FUNCTION_BLOCK DAerationLogicBasic (* Basic Function Block Type *)
  (* Standard: 61499-2 *)
  (* Version 0.0, 6/10/2026, Schneider Electric, Template *)
  PACKAGE SE.Nereda;
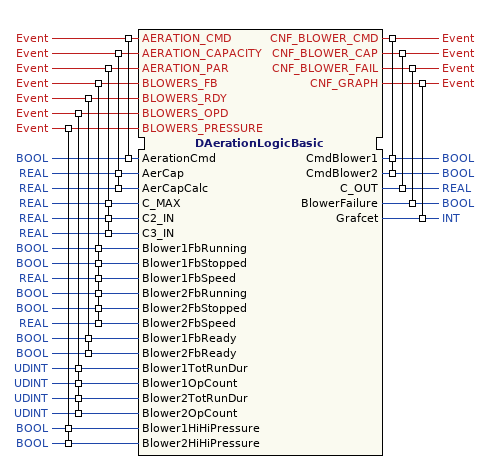
  EVENT_INPUT
    AERATION_CMD WITH AerationCmd;
    AERATION_CAPACITY WITH AerCap, AerCapCalc;
    AERATION_PAR WITH C_MAX, C2_IN, C3_IN;
    BLOWERS_FB WITH Blower1FbRunning, Blower1FbStopped, Blower1FbSpeed, Blower2FbRunning, Blower2FbStopped, Blower2FbSpeed;
    BLOWERS_RDY WITH Blower1FbReady, Blower2FbReady;
    BLOWERS_OPD WITH Blower1TotRunDur, Blower2TotRunDur, Blower1OpCount, Blower2OpCount;
    BLOWERS_PRESSURE WITH Blower1HiHiPressure, Blower2HiHiPressure;
  END_EVENT
  EVENT_OUTPUT
    CNF_BLOWER_CMD WITH CmdBlower1, CmdBlower2;
    CNF_BLOWER_CAP WITH C_OUT;
    CNF_BLOWER_FAIL WITH BlowerFailure;
    CNF_GRAPH WITH Grafcet;
  END_EVENT
  VAR_INPUT
    AerationCmd : BOOL;
    AerCap : REAL;
    AerCapCalc : REAL;
    C_MAX : REAL;
    C2_IN : REAL;
    C3_IN : REAL;
    Blower1FbRunning : BOOL;
    Blower1FbStopped : BOOL;
    Blower1FbSpeed : REAL;
    Blower2FbRunning : BOOL;
    Blower2FbStopped : BOOL;
    Blower2FbSpeed : REAL;
    Blower1FbReady : BOOL;
    Blower2FbReady : BOOL;
    Blower1TotRunDur : UDINT;
    Blower1OpCount : UDINT;
    Blower2TotRunDur : UDINT;
    Blower2OpCount : UDINT;
    Blower1HiHiPressure : BOOL;
    Blower2HiHiPressure : BOOL;
  END_VAR
  VAR_OUTPUT
    CmdBlower1 : BOOL;
    CmdBlower2 : BOOL;
    C_OUT : REAL;
    BlowerFailure : BOOL;
    Grafcet : INT;
  END_VAR
  VAR
    BL1WasRun : BOOL;
    BL2WasRun : BOOL;
  END_VAR
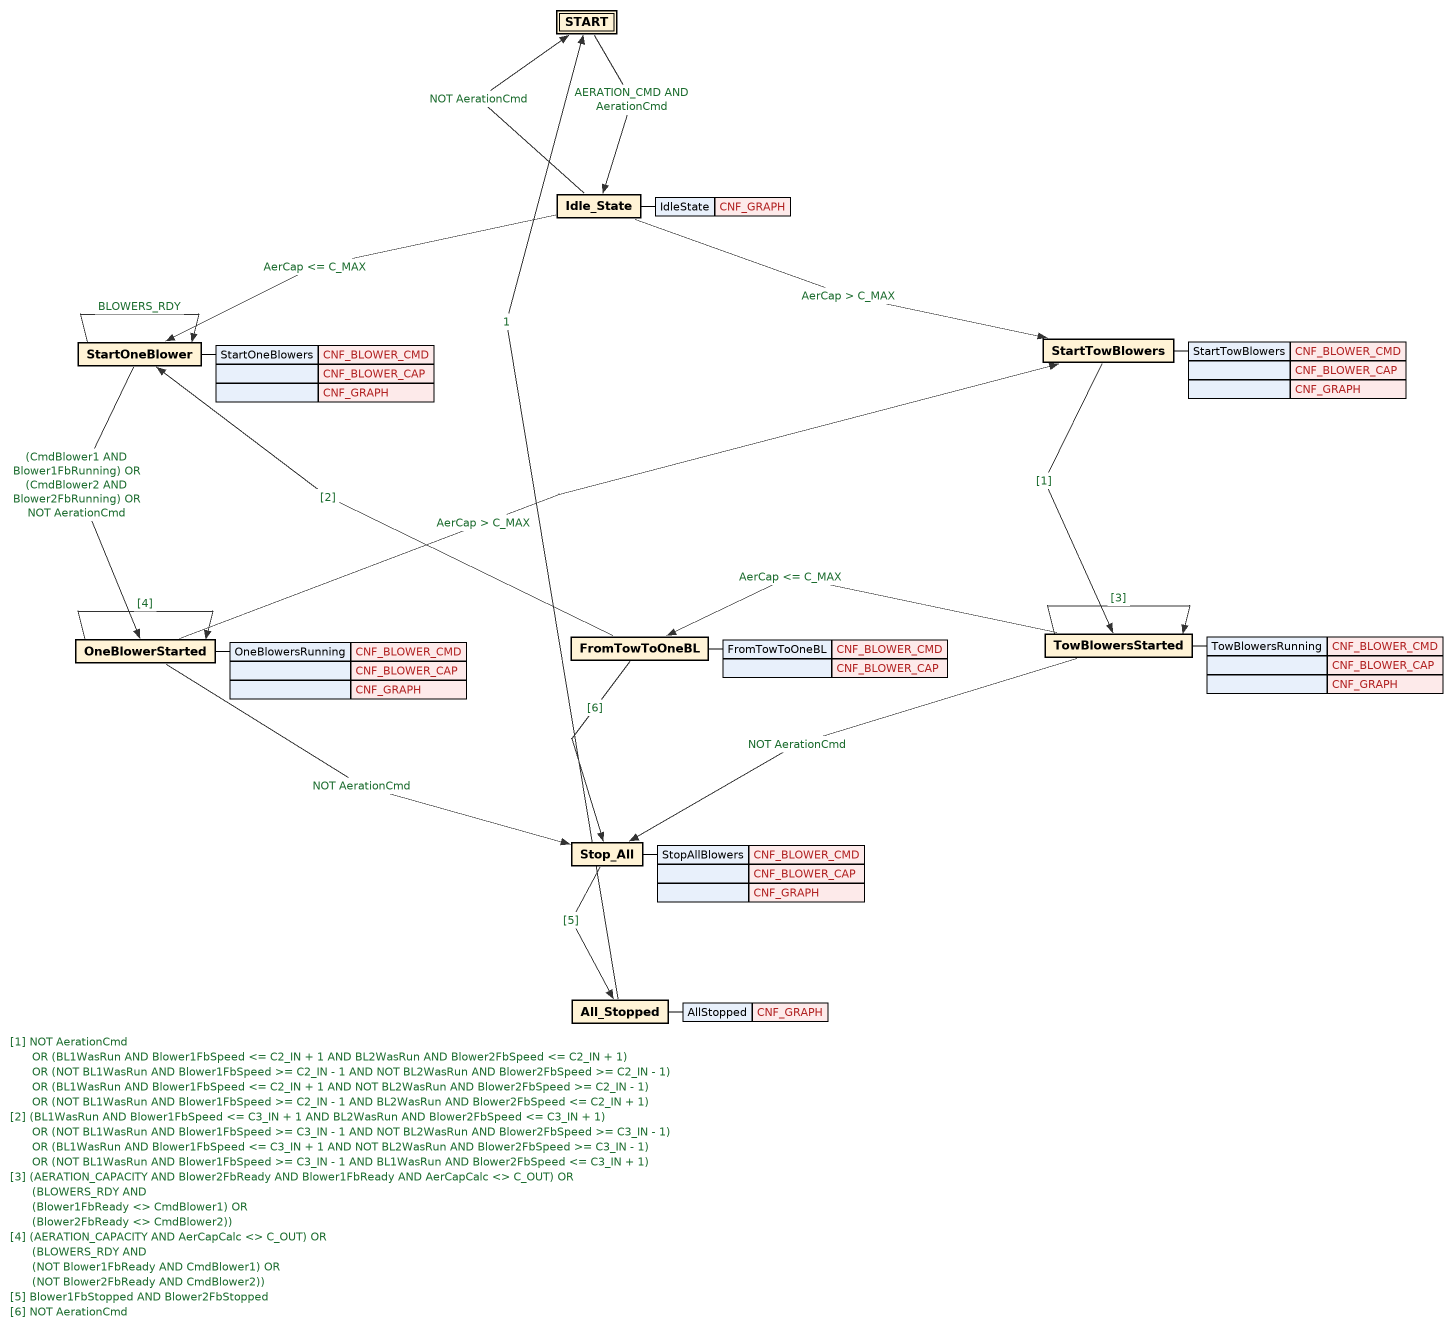
  EC_STATES
    START; (* Initial State *)
    Idle_State : IdleState -> CNF_GRAPH;
    StartTowBlowers : StartTowBlowers -> CNF_BLOWER_CMD, -> CNF_BLOWER_CAP, -> CNF_GRAPH;
    StartOneBlower : StartOneBlowers -> CNF_BLOWER_CMD, -> CNF_BLOWER_CAP, -> CNF_GRAPH;
    OneBlowerStarted : OneBlowersRunning -> CNF_BLOWER_CMD, -> CNF_BLOWER_CAP, -> CNF_GRAPH;
    TowBlowersStarted : TowBlowersRunning -> CNF_BLOWER_CMD, -> CNF_BLOWER_CAP, -> CNF_GRAPH;
    Stop_All : StopAllBlowers -> CNF_BLOWER_CMD, -> CNF_BLOWER_CAP, -> CNF_GRAPH;
    All_Stopped : AllStopped -> CNF_GRAPH;
    FromTowToOneBL : FromTowToOneBL -> CNF_BLOWER_CMD, -> CNF_BLOWER_CAP;
  END_STATES
  EC_TRANSITIONS
    START TO Idle_State := AERATION_CMD AND AerationCmd;
    Idle_State TO StartOneBlower := AerCap <= C_MAX;
    Idle_State TO StartTowBlowers := AerCap > C_MAX;
    StartOneBlower TO OneBlowerStarted := (CmdBlower1 AND Blower1FbRunning) OR (CmdBlower2 AND Blower2FbRunning) OR NOT AerationCmd;
    OneBlowerStarted TO OneBlowerStarted := (AERATION_CAPACITY AND AerCapCalc <> C_OUT) OR (BLOWERS_RDY AND (NOT Blower1FbReady AND CmdBlower1) OR (NOT Blower2FbReady AND CmdBlower2));
    StartTowBlowers TO TowBlowersStarted := NOT AerationCmd OR (BL1WasRun AND Blower1FbSpeed <= C2_IN + 1 AND BL2WasRun AND Blower2FbSpeed <= C2_IN + 1) OR (NOT BL1WasRun AND Blower1FbSpeed >= C2_IN - 1 AND NOT BL2WasRun AND Blower2FbSpeed >= C2_IN - 1) OR (BL1WasRun AND Blower1FbSpeed <= C2_IN + 1 AND NOT BL2WasRun AND Blower2FbSpeed >= C2_IN - 1) OR (NOT BL1WasRun AND Blower1FbSpeed >= C2_IN - 1 AND BL2WasRun AND Blower2FbSpeed <= C2_IN + 1);
    OneBlowerStarted TO Stop_All := NOT AerationCmd;
    TowBlowersStarted TO Stop_All := NOT AerationCmd;
    TowBlowersStarted TO FromTowToOneBL := AerCap <= C_MAX;
    All_Stopped TO START := 1;
    OneBlowerStarted TO StartTowBlowers := AerCap > C_MAX;
    TowBlowersStarted TO TowBlowersStarted := (AERATION_CAPACITY AND Blower2FbReady AND Blower1FbReady AND AerCapCalc <> C_OUT) OR (BLOWERS_RDY AND (Blower1FbReady <> CmdBlower1) OR (Blower2FbReady <> CmdBlower2));
    StartOneBlower TO StartOneBlower := BLOWERS_RDY;
    Stop_All TO All_Stopped := Blower1FbStopped AND Blower2FbStopped;
    FromTowToOneBL TO StartOneBlower := (BL1WasRun AND Blower1FbSpeed <= C3_IN + 1 AND BL2WasRun AND Blower2FbSpeed <= C3_IN + 1) OR (NOT BL1WasRun AND Blower1FbSpeed >= C3_IN - 1 AND NOT BL2WasRun AND Blower2FbSpeed >= C3_IN - 1) OR (BL1WasRun AND Blower1FbSpeed <= C3_IN + 1 AND NOT BL2WasRun AND Blower2FbSpeed >= C3_IN - 1) OR (NOT BL1WasRun AND Blower1FbSpeed >= C3_IN - 1 AND BL1WasRun AND Blower2FbSpeed <= C3_IN + 1);
    FromTowToOneBL TO Stop_All := NOT AerationCmd;
    Idle_State TO START := NOT AerationCmd;
  END_TRANSITIONS
  ALGORITHM StartOneBlowers IN ST:
;
Grafcet := 2;
// Default commands
CmdBlower1 := FALSE;
CmdBlower2 := FALSE;

// Start only one blower
IF Blower1FbReady AND NOT Blower2FbReady THEN

    // Only blower 1 is available
    CmdBlower1 := TRUE;
    CmdBlower2 := FALSE;


ELSIF Blower2FbReady AND NOT Blower1FbReady THEN

    // Only blower 2 is available
    CmdBlower1 := FALSE;
    CmdBlower2 := TRUE;


ELSIF Blower1FbReady AND Blower2FbReady THEN

    // Both blowers are available
    // First selection criteria: lowest total running duration
    IF Blower1TotRunDur < Blower2TotRunDur THEN

        CmdBlower1 := TRUE;
        CmdBlower2 := FALSE;

    ELSIF Blower2TotRunDur < Blower1TotRunDur THEN

        CmdBlower1 := FALSE;
        CmdBlower2 := TRUE;

    ELSE

        // If running durations are equal,
        // second selection criteria: lowest operation count
        IF Blower1OpCount <= Blower2OpCount THEN

            CmdBlower1 := TRUE;
            CmdBlower2 := FALSE;

        ELSE

            CmdBlower1 := FALSE;
            CmdBlower2 := TRUE;

        END_IF;

    END_IF;

ELSE

    // No blower available
    CmdBlower1 := FALSE;
    CmdBlower2 := FALSE;

END_IF;

C_OUT := C3_IN;
  END_ALGORITHM
  ALGORITHM StartTowBlowers IN ST:
;
Grafcet := 4;

CmdBlower1 := TRUE;
CmdBlower2 := TRUE;
C_OUT := C2_IN;
  END_ALGORITHM
  ALGORITHM OneBlowersRunning IN ST:
;
Grafcet := 3;

// Start only one blower
IF Blower1FbReady AND NOT Blower2FbReady THEN

	// Only blower 1 is available
	CmdBlower1 := TRUE;
	CmdBlower2 := FALSE;


ELSIF Blower2FbReady AND NOT Blower1FbReady THEN

	// Only blower 2 is available
	CmdBlower1 := FALSE;
	CmdBlower2 := TRUE;
END_IF;

// Capacity setpoint during starting
C_OUT := AerCapCalc;

BL1WasRun := Blower1FbRunning;
BL2WasRun := Blower2FbRunning;
  END_ALGORITHM
  ALGORITHM TowBlowersRunning IN ST:
;
Grafcet := 5;

// Start only one blower
IF Blower1FbReady AND NOT Blower2FbReady THEN

	// Only blower 1 is available
	CmdBlower1 := TRUE;
	CmdBlower2 := FALSE;
	C_OUT := 100;

ELSIF Blower2FbReady AND NOT Blower1FbReady THEN

	// Only blower 2 is available
	CmdBlower1 := FALSE;
	CmdBlower2 := TRUE;
	C_OUT := 100;

ELSIF Blower2FbReady AND Blower1FbReady THEN

	// Tow blowers are available
	CmdBlower1 := TRUE;
	CmdBlower2 := TRUE;
	C_OUT := AerCapCalc;
END_IF;

BL1WasRun := Blower1FbRunning;
BL2WasRun := Blower2FbRunning;
  END_ALGORITHM
  ALGORITHM StopAllBlowers IN ST:
;
Grafcet := 6;

// Default commands
CmdBlower1 := FALSE;
CmdBlower2 := FALSE;
C_OUT := 0;
  END_ALGORITHM
  ALGORITHM IdleState IN ST:
;
Grafcet := 1;
  END_ALGORITHM
  ALGORITHM AllStopped IN ST:
;
Grafcet := 7;

BL1WasRun := Blower1FbRunning;
BL2WasRun := Blower2FbRunning;
  END_ALGORITHM
  ALGORITHM FromTowToOneBL IN ST:
;
Grafcet := 8;

CmdBlower1 := TRUE;
CmdBlower2 := TRUE;
C_OUT := C3_IN;
  END_ALGORITHM
END_FUNCTION_BLOCK
